FUNCTION_BLOCK ActivateTrackForMover EXTENDS TaskBase
VAR_INPUT
END_VAR
VAR_OUTPUT
END_VAR
VAR
	mcActivateTrack : Tc3_McCollisionAvoidance.MC_ActivateTrack;
	_Axis : REFERENCE TO Tc2_MC2.AXIS_REF;
	_ActivateTrack : BOOL;
	_newTrackId : OTCID;
	_errorId: UDINT;
END_VAR

{analysis -2}

METHOD Abort : BOOL
mcActivateTrack.Execute := FALSE;
_Busy := FALSE;
_ActivateTrack := FALSE;
Abort := TRUE;
State := 0;
END_METHOD

METHOD Cycle : HRESULT
VAR_INPUT
END_VAR
Cycle := S_OK;
CASE State OF
	0:
		IF _ActivateTrack THEN
			Cycle := S_PENDING;
			_Done := FALSE;
			_Error := FALSE;
			_Busy := TRUE;
			mcActivateTrack.Execute := TRUE;
			IF mcActivateTrack.Busy THEN
				State := 10;
				_ActivateTrack := FALSE;
			END_IF
		END_IF
	
	10:
		IF NOT mcActivateTrack.Busy THEN
			IF mcActivateTrack.Done THEN
				_Done := TRUE;
				_newTrackId := mcActivateTrack.TrackId;
			ELSIF mcActivateTrack.Error THEN
				_Error := TRUE;
				_errorId := mcActivateTrack.ErrorId;
			END_IF
			_Busy := FALSE;
			mcActivateTrack.Execute := FALSE;
			State := 0;
			Cycle := S_OK;
		END_IF
	ELSE
		Cycle := E_FAIL;
END_CASE

mcActivateTrack(Axis := _Axis);
END_METHOD

METHOD PUBLIC Execute : BOOL
VAR_INPUT
	Track : OTCID;
END_VAR
IF NOT _ActivateTrack THEN
	Execute := _ActivateTrack := TRUE;
	mcActivateTrack.TrackId := Track;
ELSE
	Execute := false;
END_IF;
END_METHOD

METHOD FB_init : BOOL
VAR_INPUT
	bInitRetains : BOOL; // if TRUE, the retain variables are initialized (warm start / cold start)
	bInCopyCode : BOOL;  // if TRUE, the instance afterwards gets moved into the copy code (online change)
	Axis : reference TO AXIS_REF;
END_VAR
_Axis REF= Axis;
END_METHOD

PROPERTY PUBLIC NewTrackId : OTCID
GET
NewTrackId := _newTrackId;
END_GET
END_PROPERTY

END_FUNCTION_BLOCK

(* stored: Version 1.1.0.1
   POU ActivateTrackForMover: Id {03f53080-a7f0-4bc3-a76f-2f27947df261}, SpecialFunc None
   Method Abort: Id {12b22699-a9ca-4822-aec7-46d8d5f2084b}
   Method Cycle: Id {57b0f6ac-3d25-41af-b69c-d2ca0682dcf2}
   Method Execute: Id {b92caa48-be0c-4823-bb15-e823e8bc1934}
   Method FB_init: Id {9e9b624b-0704-4356-b4df-5729cc93ede4}
   Property NewTrackId: Id {84df412b-7c3c-4f84-98eb-ff5f562dbb1a}
   Get Get: Id {cb5898cd-640b-468a-893b-247f32481adb} *)
